{attribute 'linkalways'} 
{attribute 'no_explicit_call' := 'This FB is a CLASS and must be accessed using methods or properties'}
{attribute 'enable_dynamic_creation'}
FUNCTION_BLOCK _ETcVnFeatureDescriptorTypeAKAZE EXTENDS EnumDatatypeBase
VAR
	localData : ETcVnFeatureDescriptorTypeAKAZE;
	activeData : REFERENCE TO ETcVnFeatureDescriptorTypeAKAZE;
	enumBaseDatatype : _DINT(localData);
END_VAR

METHOD PRIVATE AddLocalEnumeration
VAR_INPUT
	Enumeration : T_MAXSTRING;
	Value : ETcVnFeatureDescriptorTypeAKAZE;
END_VAR
AddEnumeration(Enumeration, Value);
END_METHOD

PROPERTY PUBLIC Address : PVOID
GET
Address := ADR(activeData);
END_GET
END_PROPERTY

METHOD PUBLIC ClearReference
VAR_INPUT
END_VAR
activeData REF= localData;
SetBaseDatatypeReference();
END_METHOD

METHOD PUBLIC Clone : I_Datatype
VAR
    pClone : POINTER TO _ETcVnFeatureDescriptorTypeAKAZE;
END_VAR
pClone := __NEW(_ETcVnFeatureDescriptorTypeAKAZE(InitialValue := Value));
Clone := pClone^;
END_METHOD

METHOD FB_init : BOOL
VAR_INPUT
	bInitRetains : BOOL; // if TRUE, the retain variables are initialized (warm start / cold start)
	bInCopyCode : BOOL;  // if TRUE, the instance afterwards gets moved into the copy code (online change)
	InitialValue : ETcVnFeatureDescriptorTypeAKAZE;
END_VAR
localData := InitialValue;
AddBaseDatatype(enumBaseDatatype);
ClearReference();

AddLocalEnumeration('TCVN_FDT_AKAZE_KAZE_UPRIGHT', ETcVnFeatureDescriptorTypeAKAZE.TCVN_FDT_AKAZE_KAZE_UPRIGHT);
AddLocalEnumeration('TCVN_FDT_AKAZE_KAZE', ETcVnFeatureDescriptorTypeAKAZE.TCVN_FDT_AKAZE_KAZE);
AddLocalEnumeration('TCVN_FDT_AKAZE_MLDB_UPRIGHT', ETcVnFeatureDescriptorTypeAKAZE.TCVN_FDT_AKAZE_MLDB_UPRIGHT);
AddLocalEnumeration('TCVN_FDT_AKAZE_MLDB', ETcVnFeatureDescriptorTypeAKAZE.TCVN_FDT_AKAZE_MLDB);
END_METHOD

PROPERTY PUBLIC Identifier : T_MAXSTRING
GET
Identifier := 'ETcVnFeatureDescriptorTypeAKAZE';
END_GET
END_PROPERTY

METHOD IsEnumeratorValueEqual : BOOL
VAR_INPUT
	Enumerator : I_KeyValueForwardEnumerator;
END_VAR
VAR
	storedValue : ETcVnFeatureDescriptorTypeAKAZE;
END_VAR
IF NOT Enumerator.TryGet(storedValue) THEN
	RETURN;
END_IF

IsEnumeratorValueEqual := storedValue = activeData;
END_METHOD

METHOD PUBLIC MakeReferenceTo
VAR_INPUT
	ReferenceTarget : REFERENCE TO ETcVnFeatureDescriptorTypeAKAZE;
END_VAR
activeData REF= ReferenceTarget;
SetBaseDatatypeReference();
END_METHOD

METHOD PROTECTED SetBaseDatatypeReference
VAR_INPUT
END_VAR
enumBaseDatatype.MakeReferenceTo(activeData);
END_METHOD

PROPERTY PUBLIC Size : UDINT
GET
Size := SIZEOF(activeData);
END_GET
END_PROPERTY

METHOD TryMakeReferenceTo : BOOL
VAR_INPUT
	Target : I_Datatype;
END_VAR
VAR
	targetAsEnum : I_EnumDatatype;
	pTargetData : POINTER TO ETcVnFeatureDescriptorTypeAKAZE;
END_VAR
IF NOT Target.TryResolveAsEnumDatatype(targetAsEnum) THEN
	RETURN;
END_IF

IF targetAsEnum.Identifier <> Identifier THEN
	RETURN;
END_IF

pTargetData := Target.Address;
activeData REF= pTargetData^;
SetBaseDatatypeReference();
TryMakeReferenceTo := TRUE;
END_METHOD

PROPERTY PUBLIC Value : ETcVnFeatureDescriptorTypeAKAZE
GET
Value := activeData;
END_GET
SET
activeData := Value;
END_SET
END_PROPERTY

END_FUNCTION_BLOCK

(* stored: Version 1.1.0.1, ProductVersion 3.1.4024.12
   POU _ETcVnFeatureDescriptorTypeAKAZE: Id {54096076-dafc-40a0-8523-859abc409fcd}, SpecialFunc None
   Folder Constructor: Id {c2ca05cc-f622-4d07-a6f7-a2814242dff6}
   Folder Private: Id {f77a164c-15a7-4ebe-a67d-0c08c970a407}
   Folder Protected: Id {c5416a20-55cf-40bc-b61b-95b50fa86bf5}
   Method AddLocalEnumeration: Id {1dae95f7-751e-48fd-932f-33acd7033793}
   Property Address: Id {f47aa3c6-d2d2-457e-b175-c1082b60ce21}
   Get Get: Id {d85490fa-0047-40cc-82a1-5977c81099e9}
   Method ClearReference: Id {3b9eb406-6b74-4d2c-a358-dafd52e8499f}
   Method Clone: Id {75012385-8e35-4826-aad1-c414137569fe}
   Method FB_init: Id {04d2ea0c-76eb-4b26-88de-acd146c8a998}
   Property Identifier: Id {dde8a469-c8c5-4b91-942f-5517735d7efa}
   Get Get: Id {34a428eb-bf9a-48d5-ba6a-69bee0318124}
   Method IsEnumeratorValueEqual: Id {6c23b19d-413c-4632-abcc-47f5d89c6503}
   Method MakeReferenceTo: Id {4899610a-02be-4fd2-bcae-0213cb1d0376}
   Method SetBaseDatatypeReference: Id {a1dbe18f-6b2b-4bd4-80cb-9c74edd90566}
   Property Size: Id {b0cc24e0-9f3a-42b4-b32a-6392fdb48978}
   Get Get: Id {8e51e7f5-f9be-4acf-9426-1cd89c41da1c}
   Method TryMakeReferenceTo: Id {4fb5c136-5a46-418f-b822-72d01c22594f}
   Property Value: Id {cd39be42-5214-46d7-9161-761f545ce121}
   Get Get: Id {240c7ce5-992e-453c-9fbe-2d1cbb898837}
   Set Set: Id {c41d0999-c496-4861-ad7a-57a1cc3be9ef} *)
